Fanuc KAREL source: kc00028.KL

-- PROVISIONAL review KL for V770-1; original PC SHA256 936c75cce4f7c9b91233c44757d7466c19b32995b66921d8f6901bf169f5f835
-- Incomplete behavior may be omitted. Consult companion uncertainty JSON. Do not deploy.
PROGRAM KC00028
%NOLOCKGROUP
BEGIN
  -- UNRESOLVED_PC offsets 5-93; opcodes 27,22,1C,22,1C,22,1C,22,1C,22,22,22,22,1C,22,31
  -- UNRESOLVED_PC offsets 98-102; opcodes 7F
END KC00028
